FUNCTION haveDifferentIDs : BOOL
VAR_INPUT
	first: IncomingMessage;
	second: IncomingMessage;
END_VAR
VAR
END_VAR

haveDifferentIDs := (first.id.dtime <> second.id.dtime)
	OR (first.id.lowUUID <> second.id.lowUUID)
	OR (first.id.highUUID <> second.id.highUUID)
    OR (first.id.sequence <> second.id.sequence);

END_FUNCTION

(* stored: Version 1.1.0.1, ProductVersion 3.1.4022.12
   POU haveDifferentIDs: Id {1e2a1f0a-e6df-4059-9106-13397bceb00c}, SpecialFunc None *)
